# EPICS substitutions: ek9000App/Db/EL3052.substitutions
file EL3052.template
{       pattern
        {
                TERMINAL,

        }
        {
        }
}
